//{attribute 'qualified_only'}
VAR_GLOBAL
	benderLeft : FoldingMachine;
	
	robotLeft, robotRight : Robot;
	
	skidLeft, skidRight : SkidMagazine;
	magazineLeft, magazineRight : SkidMagazine;
	
	wrapper : WrapMachine;
	overhead : STRING;
	
	horizontalDriveLeft, horizontalDriveRight : ServoNC;
	verticalDriveLeft, verticalDriveRight : ClearLinkMC;
	insertionBottom : SimplePiston;
	
	innerSuctions, outerSuctions : ARRAY[Surface.TOP_LEFT..Surface.BOTTOM_RIGHT] OF SuctionPad;
END_VAR

(* stored: Version 1.1.0.1, ProductVersion 3.1.4024.11
   GVL Hardware: Id {001e16b0-c959-4c2c-800c-e6b7ef5ebc23} *)
